// Mitsubishi GX Works2 project: 0630카운터타이머   PLC: Q02/Q02H

PROGRAM MAIN
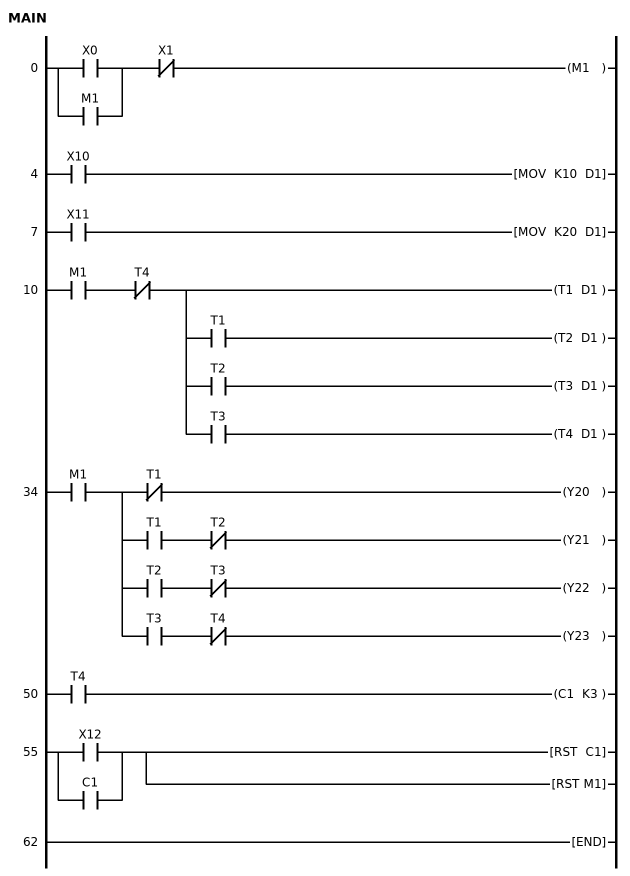
0     LD      X0
      OR      M1
      ANI     X1
      OUT     M1
4     LD      X10
      MOV     K10 D1
7     LD      X11
      MOV     K20 D1
10    LD      M1
      ANI     T4
      OUT     T1 D1
      MPS
      AND     T1
      OUT     T2 D1
      MRD
      AND     T2
      OUT     T3 D1
      MPP
      AND     T3
      OUT     T4 D1
34    LD      M1
      MPS
      ANI     T1
      OUT     Y20
      MRD
      AND     T1
      ANI     T2
      OUT     Y21
      MRD
      AND     T2
      ANI     T3
      OUT     Y22
      MPP
      AND     T3
      ANI     T4
      OUT     Y23
50    LD      T4
      OUT     C1 K3
55    LD      X12
      OR      C1
      RST     C1
      RST     M1
62    END
END_PROGRAM
